# EPICS IOC start-up script: template/scaling.iocsh
require scaling, master
scalingConfigure("scalingTest")

dbLoadRecords("/epics/base-3.15.6/require/3.1.0/siteMods/scaling/master/db/scaling.db","PREFIX=TESTSCALING,PORT=scalingTest,ADDR=0,TIMEOUT=1,MAX_ELEM=1024")
